FUNCTION_BLOCK Globals_SIFB
  (* Standard: 61499-2 *)
  (* Version 0.1, 2016-00-08, hpea485, UOA *)
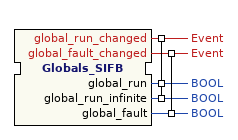
  EVENT_OUTPUT
    global_run_changed WITH global_run, global_run_infinite;
    global_fault_changed WITH global_fault;
  END_EVENT
  VAR_OUTPUT
    global_run : BOOL;
    global_run_infinite : BOOL;
    global_fault : BOOL;
  END_VAR
  VAR
    rx_global_run : BOOL; (* TOPIO_IN *)
    rx_global_run_prev : BOOL;
    rx_global_run_infinite : BOOL; (* TOPIO_IN *)
    rx_global_run_infinite_prev : BOOL;
    rx_global_fault : BOOL; (* TOPIO_IN *)
    rx_global_fault_prev : BOOL;
  END_VAR
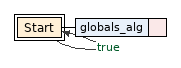
  EC_STATES
    Start : globals_alg;
  END_STATES
  EC_TRANSITIONS
    Start TO Start := true;
  END_TRANSITIONS
  ALGORITHM globals_alg IN C:
--update previous values
rx_global_run_prev <= rx_global_run;
rx_global_run_infinite_prev <= rx_global_run_infinite;
rx_global_fault_prev <= rx_global_fault;

--these are what we use to drive events
--global_run_changed_eO_alg_out;
--global_fault_changed_eO_alg_out;

if rx_global_run_prev /= rx_global_run or rx_global_run_infinite_prev /= rx_global_run_infinite then
	global_run_changed_eO_alg_out <= '1';
	global_run <= rx_global_run;
	global_run_infinite <= rx_global_run_infinite;
end if;

if rx_global_fault_prev /= rx_global_fault then
	global_fault_changed_eO_alg_out <= '1';
	global_fault <= rx_global_fault;
end if;

DONE <= '1';
  END_ALGORITHM
END_FUNCTION_BLOCK
